// Block: Coilcar_PERS

DATA_BLOCK Coilcar_PERS
VERSION : 0.1
   NON_RETAIN
   VAR
      PersistentValues : Struct
         Move : SpeedMachine_Par;
      END_STRUCT;
   END_VAR

BEGIN
   // No initialization required
END_DATA_BLOCK
